(* IEC 61131-3 sources: Workshop-4-Guevara-Prado/build, 2 files *)

(* ---- plc.st ---- *)
TYPE
  LOGLEVEL : (CRITICAL, WARNING, INFO, DEBUG) := INFO;
END_TYPE

FUNCTION_BLOCK LOGGER
  VAR_INPUT
    TRIG : BOOL;
    MSG : STRING;
    LEVEL : LOGLEVEL := INFO;
  END_VAR
  VAR
    TRIG0 : BOOL;
  END_VAR

  IF TRIG AND NOT TRIG0 THEN
  {{
   LogMessage(GetFbVar(LEVEL),(char*)GetFbVar(MSG, .body),GetFbVar(MSG, .len));
  }}
  END_IF;
  TRIG0:=TRIG;
END_FUNCTION_BLOCK

PROGRAM program0
  VAR
    A AT %IX0.0 : BOOL;
    B AT %IX0.1 : BOOL;
    C AT %IX0.2 : BOOL;
    H1 AT %QX0.0 : BOOL;
    H2 AT %QX0.1 : BOOL;
    H3 AT %QX0.2 : BOOL;
    H4 AT %QX0.3 : BOOL;
    H5 AT %QX0.4 : BOOL;
  END_VAR

  H1 := B AND A;
  H2 := B AND A OR NOT(C) AND A;
  H3 := C AND B AND A;
  H4 := NOT(C) AND NOT(B) AND NOT(A);
  H5 := B AND NOT(A) OR C AND NOT(B);
END_PROGRAM

CONFIGURATION Config0

  RESOURCE Res0 ON PLC
    TASK task0(INTERVAL := T#20ms,PRIORITY := 0);
    PROGRAM instance0 WITH task0 : program0;
  END_RESOURCE
END_CONFIGURATION

(* ---- generated_plc.st ---- *)
PROGRAM program0
  VAR
    A AT %IX0.0 : BOOL;
    B AT %IX0.1 : BOOL;
    C AT %IX0.2 : BOOL;
    H1 AT %QX0.0 : BOOL;
    H2 AT %QX0.1 : BOOL;
    H3 AT %QX0.2 : BOOL;
    H4 AT %QX0.3 : BOOL;
    H5 AT %QX0.4 : BOOL;
  END_VAR

  H1 := B AND A;
  H2 := B AND A OR NOT(C) AND A;
  H3 := C AND B AND A;
  H4 := NOT(C) AND NOT(B) AND NOT(A);
  H5 := B AND NOT(A) OR C AND NOT(B);
END_PROGRAM

CONFIGURATION Config0

  RESOURCE Res0 ON PLC
    TASK task0(INTERVAL := T#20ms,PRIORITY := 0);
    PROGRAM instance0 WITH task0 : program0;
  END_RESOURCE
END_CONFIGURATION
